KUKA KRL program: TestProfile.src, TestProfile.dat

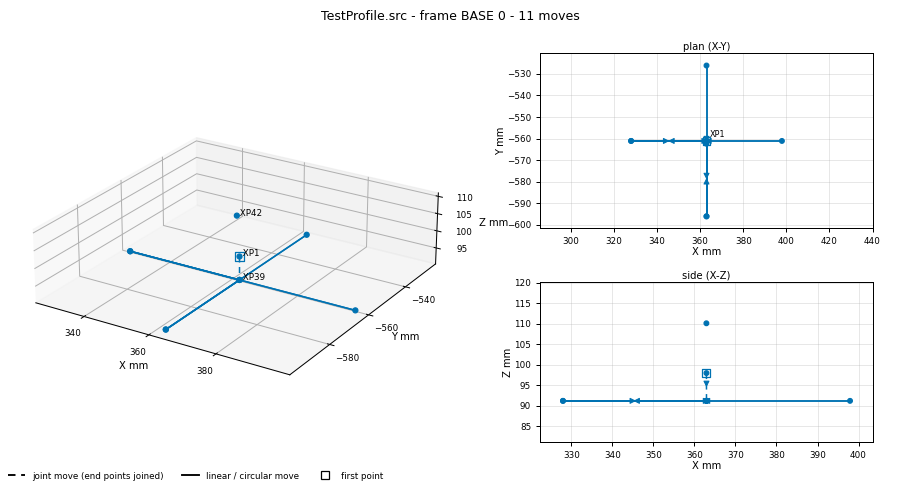
[picture p0: tool path of TestProfile.src in frame BASE 0, 11 of 12 moves have a stored position in this frame; points joined in program order, loops and branches not executed]
--- TestProfile.src ---
&ACCESS RVP
&REL 130
&PARAM TEMPLATE = C:\KRC\Roboter\Template\vorgabe
&PARAM EDITMASK = *
DEF TestProfile( )


DECL INT result, n, orient, direction, runs
DECL BOOL status
DECL FRAME RETURN_PT
DECL TORQUE_TCP_EST MyTorque


;FOLD INI
  ;FOLD BASISTECH INI
    GLOBAL INTERRUPT DECL 3 WHEN $STOPMESS==TRUE DO IR_STOPM ( )
    INTERRUPT ON 3
    BAS (#INITMOV,0 )
  ;ENDFOLD (BASISTECH INI)
  ;FOLD USER INI
    ;Make your modifications here

  ;ENDFOLD (USER INI)
;ENDFOLD (INI)
$ADVANCE = 0
$VEL.cp = 0.025
runs = 5




;Move to Hover
;FOLD PTP P1 Vel=100 % PDAT1 Tool[4]:Pneumatic_gripper Base[0];%{PE}%R 5.6.11,%MKUKATPBASIS,%CMOVE,%VPTP,%P 1:PTP, 2:P1, 3:, 5:100, 7:PDAT1
$BWDSTART=FALSE
PDAT_ACT=PPDAT1
FDAT_ACT=FP1
BAS(#PTP_PARAMS,100)
PTP XP1
;ENDFOLD

;move to approach
;FOLD PTP P39 Vel=100 % PDAT32 Tool[4]:Pneumatic_gripper Base[0];%{PE}%R 5.6.11,%MKUKATPBASIS,%CMOVE,%VPTP,%P 1:PTP, 2:P39, 3:, 5:100, 7:PDAT32
$BWDSTART=FALSE
PDAT_ACT=PPDAT32
FDAT_ACT=FP39
BAS(#PTP_PARAMS,100)
PTP XP39
;ENDFOLD


RETURN_PT = $POS_ACT_MES


;Set Parameters

status = SET_DEFAULT_IMPED()
status = SET_TOOL_FRAME(4)
status = SET_CP_STIFFNESS (4000.0, 4000.0, 100.0, 200.0, 200.0, 200.0)

;status = ENABLE_IMPEDANCE()
status = SET_CARTESIAN_FORCE( "Z",1, 0, 0, 35.0, 5000.0, -1, -1, 0.5, 0.0, 0.0, 0.0, 0.0)

status = ENABLE_CARTESIAN_FORCE()

;profile in x


;LIN_REL {Z -10}

REPEAT
MyTorque = $TORQUE_TCP_EST
UNTIL MyTorque.FT.Z >= -30

;FOLD WAIT Time=1 sec;%{PE}%R 5.6.11,%MKUKATPBASIS,%CWAIT,%VWAIT,%P 2:1
WAIT SEC 1
;ENDFOLD

;$OV_PRO = 10

LIN_REL {X -35}

FOR n = 1 TO runs STEP 1
LIN_REL {X 70}

LIN_REL {X -70}

ENDFOR

LIN_REL {X 35}

LIN_REL {Y -35}

FOR n = 1 TO runs STEP 1
LIN_REL {Y 70}

LIN_REL {Y -70}
ENDFOR

LIN_REL {Y 35}


status = DISABLE_CARTESIAN_FORCE()

$STIFFNESS.STRATEGY = 10
$STIFFNESS.COMMIT = TRUE


;$OV_PRO = 10
LIN RETURN_PT




;FOLD PTP P42 Vel=100 % PDAT35 Tool[4]:Pneumatic_gripper Base[0];%{PE}%R 5.6.11,%MKUKATPBASIS,%CMOVE,%VPTP,%P 1:PTP, 2:P42, 3:, 5:100, 7:PDAT35
$BWDSTART=FALSE
PDAT_ACT=PPDAT35
FDAT_ACT=FP42
BAS(#PTP_PARAMS,100)
PTP XP42
;ENDFOLD

END

--- TestProfile.dat ---
&ACCESS RVP
&REL 130
&PARAM TEMPLATE = C:\KRC\Roboter\Template\vorgabe
&PARAM EDITMASK = *
DEFDAT  TESTPROFILE
;FOLD EXTERNAL DECLARATIONS;%{PE}%MKUKATPBASIS,%CEXT,%VCOMMON,%P
;FOLD BASISTECH EXT;%{PE}%MKUKATPBASIS,%CEXT,%VEXT,%P
EXT  BAS (BAS_COMMAND  :IN,REAL  :IN )
DECL INT SUCCESS
;ENDFOLD (BASISTECH EXT)
;FOLD USER EXT;%{E}%MKUKATPUSER,%CEXT,%VEXT,%P
;Make here your modifications

;ENDFOLD (USER EXT)
;ENDFOLD (EXTERNAL DECLARATIONS)
DECL BASIS_SUGG_T LAST_BASIS={POINT1[] "RETURN_PT               ",POINT2[] "RETURN_PT               ",CP_PARAMS[] "CPDAT9                  ",PTP_PARAMS[] "PDAT36                  ",CONT[] "                        ",CP_VEL[] "2                       ",PTP_VEL[] "100                     ",SYNC_PARAMS[] "SYNCDAT                 ",SPL_NAME[] "S0                      "}
DECL E6POS XP1={X 362.917206,Y -561.082275,Z 97.9541626,A -0.0492787994,B -0.0317258015,C 179.964096,S 6,T 17,E1 0.000583648682,E2 0.0,E3 0.0,E4 0.0,E5 0.0,E6 0.0}
DECL FDAT FP1={TOOL_NO 4,BASE_NO 0,IPO_FRAME #BASE,POINT2[] " ",TQ_STATE FALSE}
DECL PDAT PPDAT1={VEL 100.0,ACC 100.0,APO_DIST 100.0,APO_MODE #CPTP}
DECL E6POS XP2={X 12.5678797,Y -560.598022,Z 90.5736694,A 90.0001984,B 0.00448215101,C 179.996902,S 6,T 17,E1 -0.00182819401,E2 0.0,E3 0.0,E4 0.0,E5 0.0,E6 0.0}
DECL FDAT FP2={TOOL_NO 4,BASE_NO 0,IPO_FRAME #BASE,POINT2[] " ",TQ_STATE FALSE}
DECL PDAT PPDAT2={VEL 100.0,ACC 100.0,APO_DIST 100.0,APO_MODE #CPTP}
DECL LDAT LCPDAT1={VEL 2.0,ACC 100.0,APO_DIST 100.0,APO_FAC 50.0,ORI_TYP #VAR,CIRC_TYP #BASE,JERK_FAC 50.0,EXAX_IGN 0}
DECL E6POS XP3={X 12.4056196,Y -563.239014,Z 100.730904,A 89.9864197,B -0.0702120513,C 179.992096,S 6,T 17,E1 -0.00160503399,E2 0.0,E3 0.0,E4 0.0,E5 0.0,E6 0.0}
DECL FDAT FP3={TOOL_NO 4,BASE_NO 0,IPO_FRAME #BASE,POINT2[] " ",TQ_STATE FALSE}
DECL PDAT PPDAT3={VEL 100.0,ACC 100.0,APO_DIST 100.0,APO_MODE #CPTP}
DECL PDAT PPDAT4={VEL 100.0,ACC 100.0,APO_DIST 100.0,APO_MODE #CPTP}
DECL E6POS XP4={X 13.69557,Y -563.234985,Z 167.8396,A -0.00138755003,B -0.0037752029,C -179.996704,S 6,T 17,E1 -0.00124454498,E2 0.0,E3 0.0,E4 0.0,E5 0.0,E6 0.0}
DECL FDAT FP4={TOOL_NO 4,BASE_NO 0,IPO_FRAME #BASE,POINT2[] " ",TQ_STATE FALSE}
DECL PDAT PPDAT5={VEL 100.0,ACC 100.0,APO_DIST 100.0,APO_MODE #CPTP}
DECL E6POS XP5={X -38.3249702,Y -563.137573,Z 73.9225311,A 89.9915466,B -0.0903412774,C 179.991699,S 6,T 49,E1 -0.00212001801,E2 0.0,E3 0.0,E4 0.0,E5 0.0,E6 0.0}
DECL FDAT FP5={TOOL_NO 4,BASE_NO 0,IPO_FRAME #BASE,POINT2[] " ",TQ_STATE FALSE}
DECL LDAT LCPDAT0={VEL 2.0,ACC 100.0,APO_DIST 100.0,APO_FAC 50.0,ORI_TYP #VAR,CIRC_TYP #BASE,JERK_FAC 50.0,EXAX_IGN 0}
DECL E6POS XP6={X -23.6863708,Y -563.133911,Z 73.8921432,A 89.9860229,B -0.0902003571,C 179.992203,S 6,T 49,E1 -0.00218868302,E2 0.0,E3 0.0,E4 0.0,E5 0.0,E6 0.0}
DECL FDAT FP6={TOOL_NO 4,BASE_NO 0,IPO_FRAME #BASE,POINT2[] " ",TQ_STATE FALSE}
DECL E6POS XP7={X -43.4534111,Y -563.193909,Z 74.0732269,A -0.00133702101,B -0.00409756787,C -179.988602,S 6,T 17,E1 -0.00109004998,E2 0.0,E3 0.0,E4 0.0,E5 0.0,E6 0.0}
DECL FDAT FP7={TOOL_NO 4,BASE_NO 0,IPO_FRAME #BASE,POINT2[] " ",TQ_STATE FALSE}
DECL PDAT PPDAT6={VEL 100.0,ACC 100.0,APO_DIST 100.0,APO_MODE #CPTP}
DECL E6POS XP8={X -38.3291206,Y -563.122681,Z 73.8931274,A 89.9960022,B -0.0928335115,C 179.991898,S 6,T 49,E1 -0.00218868302,E2 0.0,E3 0.0,E4 0.0,E5 0.0,E6 0.0}
DECL FDAT FP8={TOOL_NO 4,BASE_NO 0,IPO_FRAME #BASE,POINT2[] " ",TQ_STATE FALSE}
DECL PDAT PPDAT7={VEL 100.0,ACC 100.0,APO_DIST 100.0,APO_MODE #CPTP}
DECL E6POS XP9={X -38.3250084,Y -563.111328,Z 100.634003,A 89.9922638,B -0.0963689089,C 179.990601,S 6,T 49,E1 -0.00218868302,E2 0.0,E3 0.0,E4 0.0,E5 0.0,E6 0.0}
DECL FDAT FP9={TOOL_NO 4,BASE_NO 0,IPO_FRAME #BASE,POINT2[] " ",TQ_STATE FALSE}
DECL PDAT PPDAT8={VEL 100.0,ACC 100.0,APO_DIST 100.0,APO_MODE #CPTP}
DECL PDAT PPDAT9={VEL 100.0,ACC 100.0,APO_DIST 100.0,APO_MODE #CPTP}
DECL E6POS XP10={X -38.3254509,Y -563.155884,Z 100.669098,A 89.9915466,B -0.0873600096,C 179.991592,S 6,T 49,E1 -0.00218868302,E2 0.0,E3 0.0,E4 0.0,E5 0.0,E6 0.0}
DECL FDAT FP10={TOOL_NO 4,BASE_NO 0,IPO_FRAME #BASE,POINT2[] " ",TQ_STATE FALSE}
DECL PDAT PPDAT10={VEL 100.0,ACC 100.0,APO_DIST 100.0,APO_MODE #CPTP}
DECL E6POS XP11={X -38.3249702,Y -563.137573,Z 73.9225311,A 89.9915466,B -0.0903412774,C 179.991699,S 6,T 49,E1 -0.00212001801,E2 0.0,E3 0.0,E4 0.0,E5 0.0,E6 0.0}
DECL FDAT FP11={TOOL_NO 4,BASE_NO 0,IPO_FRAME #BASE,POINT2[] " ",TQ_STATE FALSE}
DECL LDAT LCPDAT2={VEL 2.0,ACC 100.0,APO_DIST 100.0,APO_FAC 50.0,ORI_TYP #VAR,CIRC_TYP #BASE,JERK_FAC 50.0,EXAX_IGN 0}
DECL E6POS XP12={X -23.6863708,Y -563.133911,Z 73.8921432,A 89.9860229,B -0.0902003571,C 179.992203,S 6,T 49,E1 -0.00218868302,E2 0.0,E3 0.0,E4 0.0,E5 0.0,E6 0.0}
DECL FDAT FP12={TOOL_NO 4,BASE_NO 0,IPO_FRAME #BASE,POINT2[] " ",TQ_STATE FALSE}
DECL PDAT PPDAT11={VEL 100.0,ACC 100.0,APO_DIST 100.0,APO_MODE #CPTP}
DECL E6POS XP13={X -38.3254509,Y -563.155884,Z 100.669098,A 89.9915466,B -0.0873600096,C 179.991592,S 6,T 49,E1 -0.00218868302,E2 0.0,E3 0.0,E4 0.0,E5 0.0,E6 0.0}
DECL FDAT FP13={TOOL_NO 4,BASE_NO 0,IPO_FRAME #BASE,POINT2[] " ",TQ_STATE FALSE}
DECL PDAT PPDAT12={VEL 100.0,ACC 100.0,APO_DIST 100.0,APO_MODE #CPTP}
DECL E6POS XP14={X -38.3249702,Y -563.137573,Z 73.9225311,A 89.9915466,B -0.0903412774,C 179.991699,S 6,T 49,E1 -0.00212001801,E2 0.0,E3 0.0,E4 0.0,E5 0.0,E6 0.0}
DECL FDAT FP14={TOOL_NO 4,BASE_NO 0,IPO_FRAME #BASE,POINT2[] " ",TQ_STATE FALSE}
DECL LDAT LCPDAT3={VEL 2.0,ACC 100.0,APO_DIST 100.0,APO_FAC 50.0,ORI_TYP #VAR,CIRC_TYP #BASE,JERK_FAC 50.0,EXAX_IGN 0}
DECL E6POS XP15={X -23.6863708,Y -563.133911,Z 73.8921432,A 89.9860229,B -0.0902003571,C 179.992203,S 6,T 49,E1 -0.00218868302,E2 0.0,E3 0.0,E4 0.0,E5 0.0,E6 0.0}
DECL FDAT FP15={TOOL_NO 4,BASE_NO 0,IPO_FRAME #BASE,POINT2[] " ",TQ_STATE FALSE}
DECL E6POS XP16={X 12.5371599,Y -609.543823,Z 100.605202,A 89.9975433,B -0.101603501,C 179.990707,S 6,T 17,E1 -0.00218868302,E2 0.0,E3 0.0,E4 0.0,E5 0.0,E6 0.0}
DECL FDAT FP16={TOOL_NO 4,BASE_NO 0,IPO_FRAME #BASE,POINT2[] " ",TQ_STATE FALSE}
DECL PDAT PPDAT13={VEL 100.0,ACC 100.0,APO_DIST 100.0,APO_MODE #CPTP}
DECL E6POS XP17={X 12.5294104,Y -619.113586,Z 73.7756195,A 89.9922714,B -0.130148306,C 179.992203,S 6,T 17,E1 -0.00255775498,E2 0.0,E3 0.0,E4 0.0,E5 0.0,E6 0.0}
DECL FDAT FP17={TOOL_NO 4,BASE_NO 0,IPO_FRAME #BASE,POINT2[] " ",TQ_STATE FALSE}
DECL PDAT PPDAT14={VEL 100.0,ACC 100.0,APO_DIST 100.0,APO_MODE #CPTP}
DECL E6POS XP18={X 12.5379105,Y -619.150574,Z 73.8089371,A 89.9952087,B -0.123240903,C 179.991592,S 6,T 17,E1 -0.00218868302,E2 0.0,E3 0.0,E4 0.0,E5 0.0,E6 0.0}
DECL FDAT FP18={TOOL_NO 4,BASE_NO 0,IPO_FRAME #BASE,POINT2[] " ",TQ_STATE FALSE}
DECL LDAT LCPDAT4={VEL 2.0,ACC 100.0,APO_DIST 100.0,APO_FAC 50.0,ORI_TYP #VAR,CIRC_TYP #BASE,JERK_FAC 50.0,EXAX_IGN 0}
DECL E6POS XP19={X 13.6944399,Y -563.275391,Z 108.710297,A -0.00195194304,B -0.00353260199,C 179.994507,S 6,T 17,E1 -0.00124454498,E2 0.0,E3 0.0,E4 0.0,E5 0.0,E6 0.0}
DECL FDAT FP19={TOOL_NO 4,BASE_NO 0,IPO_FRAME #BASE,POINT2[] " ",TQ_STATE FALSE}
DECL PDAT PPDAT15={VEL 100.0,ACC 100.0,APO_DIST 100.0,APO_MODE #CPTP}
DECL E6POS XP20={X 13.6944399,Y -563.275391,Z 108.710297,A -0.00195194304,B -0.00353260199,C 179.994507,S 6,T 17,E1 -0.00124454498,E2 0.0,E3 0.0,E4 0.0,E5 0.0,E6 0.0}
DECL FDAT FP20={TOOL_NO 4,BASE_NO 0,IPO_FRAME #BASE,POINT2[] " ",TQ_STATE FALSE}
DECL LDAT LCPDAT5={VEL 2.0,ACC 100.0,APO_DIST 100.0,APO_FAC 50.0,ORI_TYP #VAR,CIRC_TYP #BASE,JERK_FAC 50.0,EXAX_IGN 0}
DECL E6POS XP21={X -43.4534111,Y -563.193909,Z 74.0732269,A -0.00133702101,B -0.00409756787,C -179.988602,S 6,T 17,E1 -0.00109004998,E2 0.0,E3 0.0,E4 0.0,E5 0.0,E6 0.0}
DECL FDAT FP21={TOOL_NO 4,BASE_NO 0,IPO_FRAME #BASE,POINT2[] " ",TQ_STATE FALSE}
DECL PDAT PPDAT16={VEL 100.0,ACC 100.0,APO_DIST 100.0,APO_MODE #CPTP}
DECL LDAT LCPDAT6={VEL 2.0,ACC 100.0,APO_DIST 100.0,APO_FAC 50.0,ORI_TYP #VAR,CIRC_TYP #BASE,JERK_FAC 50.0,EXAX_IGN 0}
DECL E6POS XP22={X 13.6825304,Y -563.19751,Z 167.809601,A -0.00654911716,B -0.00367669109,C -179.988998,S 6,T 17,E1 -0.00109004998,E2 0.0,E3 0.0,E4 0.0,E5 0.0,E6 0.0}
DECL FDAT FP22={TOOL_NO 4,BASE_NO 0,IPO_FRAME #BASE,POINT2[] " ",TQ_STATE FALSE}
DECL PDAT PPDAT17={VEL 100.0,ACC 100.0,APO_DIST 100.0,APO_MODE #CPTP}
DECL E6POS XP23={X 11.8724298,Y -618.216309,Z 74.222847,A -178.509796,B -0.0277222507,C -179.983597,S 6,T 57,E1 -0.0177154504,E2 0.0,E3 0.0,E4 0.0,E5 0.0,E6 0.0}
DECL FDAT FP23={TOOL_NO 4,BASE_NO 0,IPO_FRAME #BASE,POINT2[] " ",TQ_STATE FALSE}
DECL LDAT LCPDAT7={VEL 2.0,ACC 100.0,APO_DIST 100.0,APO_FAC 50.0,ORI_TYP #VAR,CIRC_TYP #BASE,JERK_FAC 50.0,EXAX_IGN 0}
DECL E6POS XP24={X 11.8724298,Y -618.216309,Z 74.222847,A -178.509796,B -0.0277222507,C -179.983597,S 6,T 57,E1 -0.0177154504,E2 0.0,E3 0.0,E4 0.0,E5 0.0,E6 0.0}
DECL FDAT FP24={TOOL_NO 4,BASE_NO 0,IPO_FRAME #BASE,POINT2[] " ",TQ_STATE FALSE}
DECL LDAT LCPDAT8={VEL 2.0,ACC 100.0,APO_DIST 100.0,APO_FAC 50.0,ORI_TYP #VAR,CIRC_TYP #BASE,JERK_FAC 50.0,EXAX_IGN 0}
DECL E6POS XP25={X 12.90312,Y -587.37793,Z 126.624199,A 42.08181,B 0.664706111,C 179.027893,S 6,T 17,E1 -0.00805091858,E2 0.0,E3 0.0,E4 0.0,E5 0.0,E6 0.0}
DECL FDAT FP25={TOOL_NO 4,BASE_NO 0,IPO_FRAME #BASE,POINT2[] " ",TQ_STATE FALSE}
DECL PDAT PPDAT18={VEL 100.0,ACC 100.0,APO_DIST 100.0,APO_MODE #CPTP}
DECL E6POS XP26={X 12.90312,Y -587.37793,Z 126.624199,A 42.08181,B 0.664706111,C 179.027893,S 6,T 17,E1 -0.00805091858,E2 0.0,E3 0.0,E4 0.0,E5 0.0,E6 0.0}
DECL FDAT FP26={TOOL_NO 4,BASE_NO 0,IPO_FRAME #BASE,POINT2[] " ",TQ_STATE FALSE}
DECL PDAT PPDAT19={VEL 100.0,ACC 100.0,APO_DIST 100.0,APO_MODE #CPTP}
DECL PDAT PPDAT20={VEL 100.0,ACC 100.0,APO_DIST 100.0,APO_MODE #CPTP}
DECL E6POS XP27={X 13.6926298,Y -563.61438,Z 99.971489,A -0.00449403981,B -0.00297166291,C -179.993103,S 6,T 17,E1 -0.00139045704,E2 0.0,E3 0.0,E4 0.0,E5 0.0,E6 0.0}
DECL FDAT FP27={TOOL_NO 4,BASE_NO 0,IPO_FRAME #BASE,POINT2[] " ",TQ_STATE FALSE}
DECL E6POS XP28={X 15.5369196,Y -564.382324,Z 99.9797287,A 0.00429943902,B 0.00354765402,C -179.993698,S 6,T 17,E1 -57.84132,E2 0.0,E3 0.0,E4 0.0,E5 0.0,E6 0.0}
DECL FDAT FP28={TOOL_NO 4,BASE_NO 0,IPO_FRAME #BASE,POINT2[] " ",TQ_STATE FALSE}
DECL PDAT PPDAT21={VEL 100.0,ACC 100.0,APO_DIST 100.0,APO_MODE #CPTP}
DECL E6POS XP29={X 17.2682991,Y -564.995483,Z 99.9416733,A 0.00176301796,B 0.00983139127,C -179.987305,S 6,T 17,E1 -95.2353973,E2 0.0,E3 0.0,E4 0.0,E5 0.0,E6 0.0}
DECL FDAT FP29={TOOL_NO 4,BASE_NO 0,IPO_FRAME #BASE,POINT2[] " ",TQ_STATE FALSE}
DECL PDAT PPDAT22={VEL 100.0,ACC 100.0,APO_DIST 100.0,APO_MODE #CPTP}
DECL PDAT PPDAT23={VEL 100.0,ACC 100.0,APO_DIST 100.0,APO_MODE #CPTP}
DECL E6POS XP30={X 13.6926298,Y -563.61438,Z 99.971489,A -0.00449403981,B -0.00297166291,C -179.993103,S 6,T 17,E1 -0.00139045704,E2 0.0,E3 0.0,E4 0.0,E5 0.0,E6 0.0}
DECL FDAT FP30={TOOL_NO 4,BASE_NO 0,IPO_FRAME #BASE,POINT2[] " ",TQ_STATE FALSE}
DECL PDAT PPDAT24={VEL 100.0,ACC 100.0,APO_DIST 100.0,APO_MODE #CPTP}
DECL E6POS XP31={X 15.5369196,Y -564.382324,Z 99.9797287,A 0.00429943902,B 0.00354765402,C -179.993698,S 6,T 17,E1 -57.84132,E2 0.0,E3 0.0,E4 0.0,E5 0.0,E6 0.0}
DECL FDAT FP31={TOOL_NO 4,BASE_NO 0,IPO_FRAME #BASE,POINT2[] " ",TQ_STATE FALSE}
DECL PDAT PPDAT25={VEL 100.0,ACC 100.0,APO_DIST 100.0,APO_MODE #CPTP}
DECL E6POS XP32={X 17.2682991,Y -564.995483,Z 99.9416733,A 0.00176301796,B 0.00983139127,C -179.987305,S 6,T 17,E1 -95.2353973,E2 0.0,E3 0.0,E4 0.0,E5 0.0,E6 0.0}
DECL FDAT FP32={TOOL_NO 4,BASE_NO 0,IPO_FRAME #BASE,POINT2[] " ",TQ_STATE FALSE}
DECL PDAT PPDAT26={VEL 100.0,ACC 100.0,APO_DIST 100.0,APO_MODE #CPTP}
DECL E6POS XP33={X 13.6926298,Y -563.61438,Z 99.971489,A -0.00449403981,B -0.00297166291,C -179.993103,S 6,T 17,E1 -0.00139045704,E2 0.0,E3 0.0,E4 0.0,E5 0.0,E6 0.0}
DECL FDAT FP33={TOOL_NO 4,BASE_NO 0,IPO_FRAME #BASE,POINT2[] " ",TQ_STATE FALSE}
DECL PDAT PPDAT27={VEL 100.0,ACC 100.0,APO_DIST 100.0,APO_MODE #CPTP}
DECL E6POS XP34={X 15.5369196,Y -564.382324,Z 99.9797287,A 0.00429943902,B 0.00354765402,C -179.993698,S 6,T 17,E1 -57.84132,E2 0.0,E3 0.0,E4 0.0,E5 0.0,E6 0.0}
DECL FDAT FP34={TOOL_NO 4,BASE_NO 0,IPO_FRAME #BASE,POINT2[] " ",TQ_STATE FALSE}
DECL PDAT PPDAT28={VEL 100.0,ACC 100.0,APO_DIST 100.0,APO_MODE #CPTP}
DECL E6POS XP35={X 17.2682991,Y -564.995483,Z 99.9416733,A 0.00176301796,B 0.00983139127,C -179.987305,S 6,T 17,E1 -95.2353973,E2 0.0,E3 0.0,E4 0.0,E5 0.0,E6 0.0}
DECL FDAT FP35={TOOL_NO 4,BASE_NO 0,IPO_FRAME #BASE,POINT2[] " ",TQ_STATE FALSE}
DECL PDAT PPDAT29={VEL 100.0,ACC 100.0,APO_DIST 100.0,APO_MODE #CPTP}
DECL E6POS XP36={X 13.6926298,Y -563.61438,Z 99.971489,A -0.00449403981,B -0.00297166291,C -179.993103,S 6,T 17,E1 -0.00139045704,E2 0.0,E3 0.0,E4 0.0,E5 0.0,E6 0.0}
DECL FDAT FP36={TOOL_NO 4,BASE_NO 0,IPO_FRAME #BASE,POINT2[] " ",TQ_STATE FALSE}
DECL PDAT PPDAT30={VEL 100.0,ACC 100.0,APO_DIST 100.0,APO_MODE #CPTP}
DECL E6POS XP37={X 15.5369196,Y -564.382324,Z 99.9797287,A 0.00429943902,B 0.00354765402,C -179.993698,S 6,T 17,E1 -57.84132,E2 0.0,E3 0.0,E4 0.0,E5 0.0,E6 0.0}
DECL FDAT FP37={TOOL_NO 4,BASE_NO 0,IPO_FRAME #BASE,POINT2[] " ",TQ_STATE FALSE}
DECL PDAT PPDAT31={VEL 100.0,ACC 100.0,APO_DIST 100.0,APO_MODE #CPTP}
DECL E6POS XP38={X 17.2682991,Y -564.995483,Z 99.9416733,A 0.00176301796,B 0.00983139127,C -179.987305,S 6,T 17,E1 -95.2353973,E2 0.0,E3 0.0,E4 0.0,E5 0.0,E6 0.0}
DECL FDAT FP38={TOOL_NO 4,BASE_NO 0,IPO_FRAME #BASE,POINT2[] " ",TQ_STATE FALSE}
DECL PDAT PPDAT32={VEL 100.0,ACC 100.0,APO_DIST 100.0,APO_MODE #CPTP}
DECL E6POS XP39={X 362.931213,Y -561.104309,Z 91.1815872,A -0.0495438501,B -0.0349056087,C 179.959106,S 6,T 17,E1 0.000583648682,E2 0.0,E3 0.0,E4 0.0,E5 0.0,E6 0.0}
DECL FDAT FP39={TOOL_NO 4,BASE_NO 0,IPO_FRAME #BASE,POINT2[] " ",TQ_STATE FALSE}
DECL PDAT PPDAT33={VEL 100.0,ACC 100.0,APO_DIST 100.0,APO_MODE #CPTP}
DECL E6POS XP40={X 15.5369196,Y -564.382324,Z 99.9797287,A 0.00429943902,B 0.00354765402,C -179.993698,S 6,T 17,E1 -57.84132,E2 0.0,E3 0.0,E4 0.0,E5 0.0,E6 0.0}
DECL FDAT FP40={TOOL_NO 4,BASE_NO 0,IPO_FRAME #BASE,POINT2[] " ",TQ_STATE FALSE}
DECL PDAT PPDAT34={VEL 100.0,ACC 100.0,APO_DIST 100.0,APO_MODE #CPTP}
DECL E6POS XP41={X 17.2682991,Y -564.995483,Z 99.9416733,A 0.00176301796,B 0.00983139127,C -179.987305,S 6,T 17,E1 -95.2353973,E2 0.0,E3 0.0,E4 0.0,E5 0.0,E6 0.0}
DECL FDAT FP41={TOOL_NO 4,BASE_NO 0,IPO_FRAME #BASE,POINT2[] " ",TQ_STATE FALSE}
DECL PDAT PPDAT35={VEL 100.0,ACC 100.0,APO_DIST 100.0,APO_MODE #CPTP}
DECL E6POS XP42={X 362.904388,Y -562.374207,Z 110.094101,A -0.0444133505,B -0.02433943,C 179.973907,S 6,T 17,E1 0.0001459122,E2 0.0,E3 0.0,E4 0.0,E5 0.0,E6 0.0}
DECL FDAT FP42={TOOL_NO 4,BASE_NO 0,IPO_FRAME #BASE,POINT2[] " ",TQ_STATE FALSE}
DECL E6POS XRETURN_PT={X -52.0832787,Y -581.914124,Z 247.525101,A 1.37840497,B -2.5678699,C -177.104996,S 6,T 17,E1 1.12184095,E2 0.0,E3 0.0,E4 0.0,E5 0.0,E6 0.0}
DECL FDAT FRETURN_PT={TOOL_NO 4,BASE_NO 0,IPO_FRAME #BASE,POINT2[] " ",TQ_STATE FALSE}
DECL LDAT LCPDAT9={VEL 2.0,ACC 100.0,APO_DIST 100.0,APO_FAC 50.0,ORI_TYP #VAR,CIRC_TYP #BASE,JERK_FAC 50.0,EXAX_IGN 0}
DECL PDAT PPDAT36={VEL 100.0,ACC 100.0,APO_DIST 100.0,APO_MODE #CPTP}
ENDDAT
